{attribute 'GeneratedUsingTerminal: EL6692-0002-0016'}
{attribute addProperty BoxType "EL6692-0002-0016"}
{attribute addProperty Id "SYNC_InputsAT %I*SYNC_Inputs_462ED3216IO_InputsEMPTY_STRUCTURE0IO_OutputsEMPTY_STRUCTURE0WcStateAT %I*WcState_9091E0EB2InfoDataAT %I*InfoData_90184F0C16"}
{attribute addProperty CRC "4046274739"}
{attribute addProperty Size "24"}
TYPE EL6692_F12D40B3 EXTENDS EtcSlaveTerminalBase_947E5A46 :
STRUCT
	{attribute addProperty Name "SYNC_Inputs"}
	SYNC_Inputs : SYNC_Inputs_462ED321;
	{attribute addProperty Name "IO_Inputs"}
	IO_Inputs : EMPTY_STRUCTURE;
	{attribute addProperty Name "IO_Outputs"}
	IO_Outputs : EMPTY_STRUCTURE;
	{attribute addProperty Name "WcState"}
	WcState : WcState_9091E0EB;
	{attribute addProperty Name "InfoData"}
	InfoData : InfoData_90184F0C;
END_STRUCT
END_TYPE

(* stored: Version 1.2.0.0, ProductVersion 3.1.4024.9
   DUT EL6692_F12D40B3: Id {4f47fab8-2b99-4b75-8850-9a41e0c5517d} *)
